FUNCTION "LAxisCtrl_UnpubEmergencyDecSpeedAxis" : LReal
{ S7_Optimized_Access := 'TRUE' }
AUTHOR : 'tech.team.motioncontrol@siemens.com'
FAMILY : AxisCtrl
VERSION : 1.1
   VAR_INPUT
      axis {InstructionName := 'TO_SpeedAxis'; LibVersion := '5.0'} : TO_SpeedAxis;
   END_VAR


BEGIN
	// Read axis parameter
	#LAxisCtrl_UnpubEmergencyDecSpeedAxis := #axis.DynamicDefaults.EmergencyDeceleration;
END_FUNCTION

